KUKA KRL program: start_weld_respot.src

&ACCESS RVO
&REL 149
&COMMENT start_weld_RESPOT
&PARAM DISKPATH = KRC:\R1\Program\SubRotinas
DEF start_weld_RESPOT( )
;
;FOLD OUT 3333 'R1 trabalho concluído' State=FALSE ;%{PE}%R 8.2.20,%MKUKATPBASIS,%COUT,%VOUTX,%P 2:3333, 3:R1 trabalho concluído, 5:FALSE, 6:
$OUT[3333]=FALSE
;ENDFOLD
;
END
